{attribute 'TcGenerated'}
// This function has been automatically generated from the project information.
VAR_GLOBAL CONSTANT
	{attribute 'const_non_replaced'}
	{attribute 'linkalways'}
	stLibVersion_Vacuum_System_Simulator_Library : ST_LibVersion := (iMajor := 1, iMinor := 0, iBuild := 0, iRevision := 0, sVersion := '1.0.0');
END_VAR

(* stored: Version 1.1.0.1, ProductVersion 3.1.4020.12
   GVL Global_Version: Id b7a03291-ec7c-448c-ad3d-d896c9b9cdef *)
